// TIA Portal V18 export
DATA_BLOCK "DB_DI"   // DB1
{ S7_Optimized_Access := 'FALSE' }
VERSION : 0.1
// stored: AutoNumber true, DBAccessibleFromOPCUA true, DBAccessibleFromWebserver true, IsOnlyStoredInLoadMemory false, IsWriteProtectedInAS false
   VAR
      in_SelStart : Bool;
      in_SelStop : Bool;
      in_BtnEmergency : Bool;
      in_BtnReset : Bool;
      in_Capacitive : Bool;
      in_5 : Bool;
      in_6 : Bool;
      in_PhCell_0 : Bool;
      in_PhCell_1 : Bool;
      in_PhCell_2 : Bool;
      in_PhCell_3 : Bool;
      in_PhCell_4 : Bool;
      in_PhCell_5 : Bool;
      in_PhCell_6 : Bool;
      in_PhCell_7 : Bool;
      in_PhCell_8 : Bool;
      in_Picker : Bool;
      in_17 : Bool;
      in_18 : Bool;
      in_19 : Bool;
      in_20 : Bool;
      in_21 : Bool;
      in_22 : Bool;
      in_23 : Bool;
      in_24 : Bool;
      in_25 : Bool;
      in_26 : Bool;
      in_27 : Bool;
      in_28 : Bool;
      in_29 : Bool;
      in_30 : Bool;
      in_31 : Bool;
      BtnReset_p : Bool;
      PhCell_0_p : Bool;
      PhCell_0_n : Bool;
      PhCell_1_p : Bool;
      PhCell_1_n : Bool;
      PhCell_2_p : Bool;
      PhCell_2_n : Bool;
      PhCell_3_p : Bool;
      PhCell_3_n : Bool;
      PhCell_4_p : Bool;
      PhCell_4_n : Bool;
      PhCell_5_p : Bool;
      PhCell_5_n : Bool;
      PhCell_6_p : Bool;
      PhCell_6_n : Bool;
      PhCell_7_p : Bool;
      PhCell_7_n : Bool;
      PhCell_8_p : Bool;
      PhCell_8_n : Bool;
   END_VAR
BEGIN
END_DATA_BLOCK
